Universal Robots PolyScope program: Timer.urp

ProgramRoot directory=/home/ur/ursim-3.1/programs; kinematics=(a=[0, -0.425, -0.39225, 0, 0, 0], d=[0.08916, 0, 0, 0.10915, 0.09465, 0.0823], alpha=[1.5708, 0, 0, 1.5708, -1.5708, 0], deltaTheta=[0, 0, 0, 0, 0, 0], status=notInitialized); lastSavedInVersion=(project__name=Polyscope, major__version=3, minor__version=1, svn__revision=17195, build__date=Mar 11 2015, 13:02:28); name=Timer; programVersion=(project__name=Polyscope, major__version=3, minor__version=1, svn__revision=17195, build__date=Mar 11 2015, 13:02:28); robotEnvironmentFileName=default; serialNumberRobot=2014350001
  BeforeStart description=COMMAND_SEQUENCE_BEFORE_PROGRAM_START; name=BeforeStart
    Assignment expr=True; operatorValueType=INTEGER; valueSource=EXPRESSION
    Assignment expr=0; operatorValueType=INTEGER; valueSource=EXPRESSION
  MainProgram cartesianAcceleration=1.2; cartesianSpeed=0.25; jointAcceleration=1.3962634015954636; jointSpeed=1.0471975511965976; sharedProcessMoveBlendRadius=0.025; motionType=JOINT_SPACE; runOnlyOneCycle=true
    Wait 
    Assignment expr=False; operatorValueType=INTEGER; valueSource=EXPRESSION
    Wait 
    Assignment expr=True; operatorValueType=INTEGER; valueSource=EXPRESSION
  Thread name=Thread_1
    If expr=ExpressionVariableNode≟ False; type=IF_NODE
      Assignment expr=ExpressionVariableNode+0.01; operatorValueType=INTEGER; valueSource=EXPRESSION
    Wait 
